(* PLC project LibIT_STEPPER_MOTOR, lamsystems-it.ru LibIT_STEPPER_MOTOR 1 *)
(* stored: creationDateTime 2019-11-13T09:37:45, productRelease 0, modificationDateTime 2023-01-20T15:46:21, version 1 *)

(* Статус шагового двигателя *)
FUNCTION_BLOCK StepStatus
  VAR_INPUT
    DOnStep : BYTE := 0;  (* номер выхода *)
    DOnDir : BYTE := 0;  (* номер выхода *)
  END_VAR
  VAR_OUTPUT
    State : BYTE := 0;  (* код результата исполнения блока *)
    Ok : BYTE := 0;  (* код результата исполнения блока *)
  END_VAR

            {extern void App_StepperStatus(STEPSTATUS*);App_StepperStatus(data__);}

          
END_FUNCTION_BLOCK

(* Запуск шагового двигателя *)
FUNCTION_BLOCK StepMotor
  VAR_INPUT
    Ex : BOOL := FALSE;  (* разрешение на выполнение *)
    Rst : BOOL := FALSE;  (* сброс счетчика шагов *)
    Stop : BYTE := 0;  (* остановка мотора *)
    DOnStep : BYTE := 0;  (* номер выхода step *)
    DOnDir : BYTE := 0;  (* номер выхода dir *)
    StartSpeed : WORD := 0;  (* стартовая скорость *)
    Speed : WORD := 0;  (* скорость *)
    AcN : WORD := 0;  (* кол-во шагов ускорения *)
    DecN : WORD := 0;  (* кол-во шагов остановки *)
    Steps : DWORD := 0;  (* кол-во шагов *)
    Dir : BOOL := FALSE;  (* направление вращения *)
    Dir_delay : WORD := 0;  (* задержка смены направления вращения *)
    StepRPM : WORD := 0;  (* кол-во шагов на оборот *)
    DivStep : WORD := 0;  (* деление шага (микрошаг) *)
  END_VAR
  VAR_OUTPUT
    Ok : BYTE := 0;  (* код результата исполнения блока *)
    State : BYTE := 0;  (* статус двигателя *)
    Err : BYTE := 0;  (* код ошибки исполнения блока *)
  END_VAR

            {extern void App_StepperMove(STEPMOTOR*);App_StepperMove(data__);}

          
END_FUNCTION_BLOCK
